// TIA Portal V20 export
DATA_BLOCK "CommsProcessData"   // DB205
   VAR
      CommsErrorStatus : Word;
      DbErrorStatus : Word;
      DataLoaded : Bool;
      SequenceStep : USInt;
      SequenceIndex : USInt;
      CommsFault : Bool;
      CommsFaultOneShot : Bool;
      CommsResetPulse : Bool;
      NodeFaultCount : Array[0..14] of Int;
      NodeFault : Array[0..14] of Bool;
      SequenceComplete : Bool;
      ConfigWord : Word := 16#041F;
   END_VAR
BEGIN
END_DATA_BLOCK
